FUNCTION_BLOCK FaultDiagnosis (* Fault Diagnosis Function Block *)
  (* Standard: 61499-2 *)
  (* Version 1.0, Example Corp *)
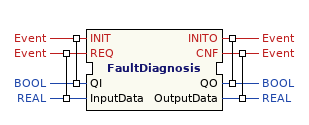
  EVENT_INPUT
    INIT WITH QI; (* Initialization Request *)
    REQ WITH InputData; (* Normal Execution Request *)
  END_EVENT
  EVENT_OUTPUT
    INITO WITH QO; (* Initialization Confirm *)
    CNF WITH OutputData; (* Execution Confirmation *)
  END_EVENT
  VAR_INPUT
    QI : BOOL; (* Input event qualifier *)
    InputData : REAL; (* Input data *)
  END_VAR
  VAR_OUTPUT
    QO : BOOL; (* Output event qualifier *)
    OutputData : REAL; (* Output data *)
  END_VAR
  EC_STATES
    START; (* Initial State *)
    INIT : INIT -> INITO; (* Initialization *)
    REQ : REQ -> CNF; (* Normal execution *)
  END_STATES
  ALGORITHM INIT IN ST: (* Initialization algorithm *)
QO := QI;
  END_ALGORITHM
  ALGORITHM REQ IN ST: (* Normal execution algorithm *)
OutputData := InputData * 2.0;
  END_ALGORITHM
END_FUNCTION_BLOCK
